{attribute 'qualified_only'}
{attribute 'to_string'}
TYPE EXCEPTION_CATCH_POINT :
(
	BEFORE_EXECUTE,
	AFTER_EXECUTE,
	BEFORE_EXECUTE_PLUGINS,
	BEFORE_CHILDREN_WORKING,
	AFTER_CHILDREN_WORKING,
	BEFORE_CHILDREN_STOPPED,
	AFTER_CHILDREN_STOPPED,
	BEFORE_CHILDREN_RESET,
	AFTER_CHILDREN_RESET,
	RECOVER,
	PROCESS_INPUT,
	PROCESS_OUTPUT,
	BEFORE_CHILDREN_PROCESS_INPUT,
	AFTER_CHILDREN_PROCESS_INPUT,
	BEFORE_CHILDREN_PROCESS_OUTPUT,
	AFTER_CHILDREN_PROCESS_OUTPUT,
	AFTER_EXECUTE_PLUGINS,
	USER_DEFINED
);
END_TYPE

(* stored: Version 1.1.0.1
   DUT EXCEPTION_CATCH_POINT: Id {ad81853c-05dd-4304-b0e6-7e0ebe43d4f0} *)
